// TIA Portal V19 export
DATA_BLOCK "DATE&TIME"   // DB8
{ S7_Optimized_Access := 'TRUE' }
// stored: MemoryReserve 100
   VAR RETAIN
      "RET READ" : Int;
      "RET WRITE" : Int;
      WRITE_DAY : Int;
      WRITE_MONTH : Int;
      WRITE_YEAR : Int;
      WRITE_HOUR : Int;
      WRITE_MINUTE : Int;
      WRITE_SECOND : Int;
      "READ RE" : DTL;
      "WRITE RE" : DTL;
      SET_DTM : Bool;
   END_VAR
BEGIN
END_DATA_BLOCK
